{attribute 'pack_mode' := '1'}
TYPE TRunDataVision :
STRUCT
		iUseModel		: INT;
		iMaxModel		: INT;
		TVisionPartData	: TVisionPartData;
END_STRUCT
END_TYPE

(* stored: Version 1.1.0.1, ProductVersion 3.1.4022.12
   DUT TRunDataVision: Id {fdf05332-99d5-40b6-9334-8c2d0e9bd0af} *)
